TYPE E_StepPrimaryCriterion : (
    STEP_CRIT_RELATIVE_DISTANCE := 0,
    STEP_CRIT_STEP_TIME := 10,
    STEP_CRIT_FORCE_DECLINE_TO := 20
); END_TYPE

(* stored: Version 1.1.0.1
   DUT E_StepPrimaryCriterion: Id {E3000000-0000-4000-8000-000000000010} *)
